// TIA Portal V17 export
// export: Created 2022-10-14T12:26:42.9399606Z, ExportSetting WithDefaults, DisplayName Totally Integrated Automation Portal, DisplayVersion V17 Update 4, DisplayName TIA Portal Openness, DisplayVersion V17 Update 4, DisplayName TIA Portal Version Control Interface, DisplayVersion V17, DisplayName SINAMICS Startdrive Advanced, DisplayVersion V17 Update2, DisplayName SINAMICS Startdrive G130, G150, S120, S150, SINAMICS MV, S210, DisplayVersion V17 Update2, DisplayName SINAMICS Startdrive G110M, G120, G120C, G120D, G120P, G115D, DisplayVersion V17 Update2, DisplayName STEP 7 Professional, DisplayVersion V17 Update 4, DisplayName STEP 7 Safety, DisplayVersion V17, DisplayName WinCC Advanced / Unified PC, DisplayVersion V17 Update 4
FUNCTION_BLOCK "1002_Device"   // FB1002, FBD
{ S7_Optimized_Access := 'TRUE' }
VERSION : 0.1
// Bender-gerät kommunikation baustein (COM465ID)
//                               FEST GmbH  
//  M.Alsouki            27.11.2019     v 1.04
// stored: AutoNumber false, IsIECCheckEnabled false, IsRetainMemResEnabled false, MemoryReserve 100, SetENOAutomatically false, UDAEnableTagReadback false
   VAR_INPUT
      Takt : Bool;
      HW_RCV : HW_SUBMODULE;
      HW_SND : HW_SUBMODULE;
      Addr : Array[1.."DeviceNr"] of Byte;
      Gruppen : Array[1.."DeviceNr"] of "Channels";
      "Message-Typ" : Byte := b#01;
      SubSysAdr : Byte := b#01;
   END_VAR
   VAR_OUTPUT
      Devices : Array[1.."DeviceNr"] of "Dates_Pro_Channel";
   END_VAR
   VAR
      HAdr { S7_SetPoint := 'True'} : Byte;
      HKanal : Byte;
      SND_ID : Byte;
      RCV_ID : Byte;
      Data_RCV : "RCV_Dates";
      i : Byte := 1;
      K : Int := 1;
      AA : Int := 1;
      HM1 : Bool;
      HM2 : Bool;
      HM3 : Bool;
      HM4 : Bool;
      RESET_AA : Int;
      RESET_i : Int;
      RESET_i_Byte : USInt;
   END_VAR
   VAR_TEMP
      ERROR : Bool;
   END_VAR
   // Gruppen[1].Kanal[1] := 16#01;
   // Gruppen[1].Kanal[2] := 16#02;
   // Gruppen[1].Kanal[3] := 16#03;
   // Gruppen[1].Kanal[4] := 16#04;
   // Gruppen[2].Kanal[1] := 16#01;
   // Gruppen[2].Kanal[2] := 16#02;
   // Gruppen[2].Kanal[3] := 16#03;
   // Gruppen[2].Kanal[4] := 16#04;
   // Gruppen[3].Kanal[1] := 16#01;
   // Gruppen[3].Kanal[2] := 16#02;
   // Gruppen[3].Kanal[3] := 16#03;
   // Gruppen[3].Kanal[4] := 16#04;
   // Gruppen[4].Kanal[1] := 16#01;
   // Gruppen[4].Kanal[2] := 16#02;
   // Gruppen[4].Kanal[3] := 16#03;
   // Gruppen[4].Kanal[4] := 16#04;
   // Gruppen[5].Kanal[1] := 16#05;
   // Gruppen[5].Kanal[2] := 16#06;
   // Gruppen[5].Kanal[3] := 16#07;
   // Gruppen[5].Kanal[4] := 16#08;
   // Gruppen[6].Kanal[1] := 16#09;
   // Gruppen[6].Kanal[2] := 16#0a;
   // Gruppen[6].Kanal[3] := 16#0b;
   // Gruppen[6].Kanal[4] := 16#0c;
   VAR_TEMP   // added for the SCL form of the ladder/FBD networks
      _w1 : Bool;
      _w2 : Bool;
   END_VAR
BEGIN

REGION Network 1
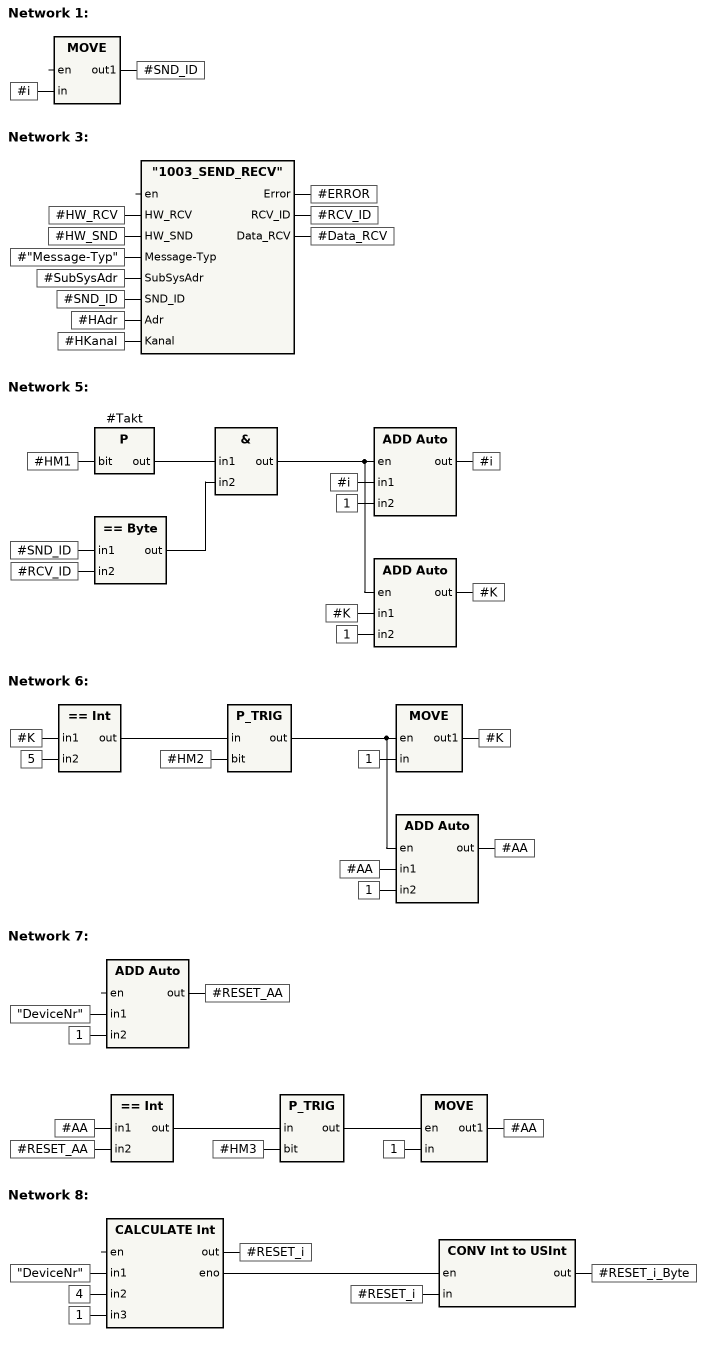
   #SND_ID := #i;
END_REGION

REGION Network 2 (SCL)
   #HAdr := #Addr[#AA];
   #HKanal := #Gruppen[#AA].Kanal[#K];
END_REGION

REGION Network 3
   "1003_SEND_RECV"(HW_RCV := #HW_RCV,
                    HW_SND := #HW_SND,
                    "Message-Typ" := #"Message-Typ",
                    SubSysAdr := #SubSysAdr,
                    SND_ID := #SND_ID,
                    Adr := #HAdr,
                    Kanal := #HKanal,
                    Error => #ERROR,
                    RCV_ID => #RCV_ID,
                    Data_RCV => #Data_RCV);
END_REGION

REGION Network 4 (SCL)
   #Devices[#AA].Kanal[#K] := #Data_RCV;
END_REGION

REGION Network 5
   // i: ID index
   // K: Kanal index
   #_w1 := #Takt AND NOT #HM1;   // rising edge of #Takt
   #HM1 := #Takt;
   IF #_w1 AND (#SND_ID = #RCV_ID) THEN
       #i := #i + 1;
       #K := #K + 1;
   END_IF;
END_REGION

REGION Network 6
   // AA:  Adresse index
   #_w1 := #K = 5;
   #_w2 := #_w1 AND NOT #HM2;   // rising edge
   #HM2 := #_w1;
   IF #_w2 THEN
       #K := 1;
       #AA := #AA + 1;
   END_IF;
END_REGION

REGION Network 7
   #RESET_AA := "DeviceNr" + 1;
   #_w1 := #AA = #RESET_AA;
   #_w2 := #_w1 AND NOT #HM3;   // rising edge
   #HM3 := #_w1;
   IF #_w2 THEN #AA := 1; END_IF;
END_REGION

REGION Network 8
   #RESET_i := ("DeviceNr"*4)+1;
   #RESET_i_Byte := INT_TO_USINT(#RESET_i);
END_REGION

REGION Network 9
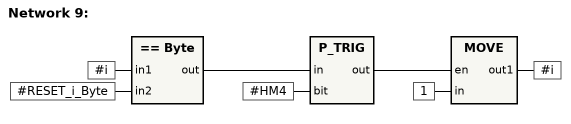
   #_w1 := #i = #RESET_i_Byte;
   #_w2 := #_w1 AND NOT #HM4;   // rising edge
   #HM4 := #_w1;
   IF #_w2 THEN #i := 1; END_IF;
END_REGION
END_FUNCTION_BLOCK
